% RSLogix 500 project I2P HANDS-ON 3 - LEO.RSS, saved by version 10.00.00.00 %
PROJECT "ML04B"    % processor: Bul.1763 MicroLogix 1100 Series B %

PROGRAM FILES
  LAD 2   10 rungs

DATA FILES
  O0 OUTPUT  4 elements
  I1 INPUT  6 elements
  S2 STATUS  66 elements
  B3 BINARY  1 elements
  T4 TIMER  1 elements
  C5 COUNTER  1 elements
  R6 CONTROL  1 elements
  N7 INTEGER  1 elements
  F8 FLOAT  1 elements

LADDER 2
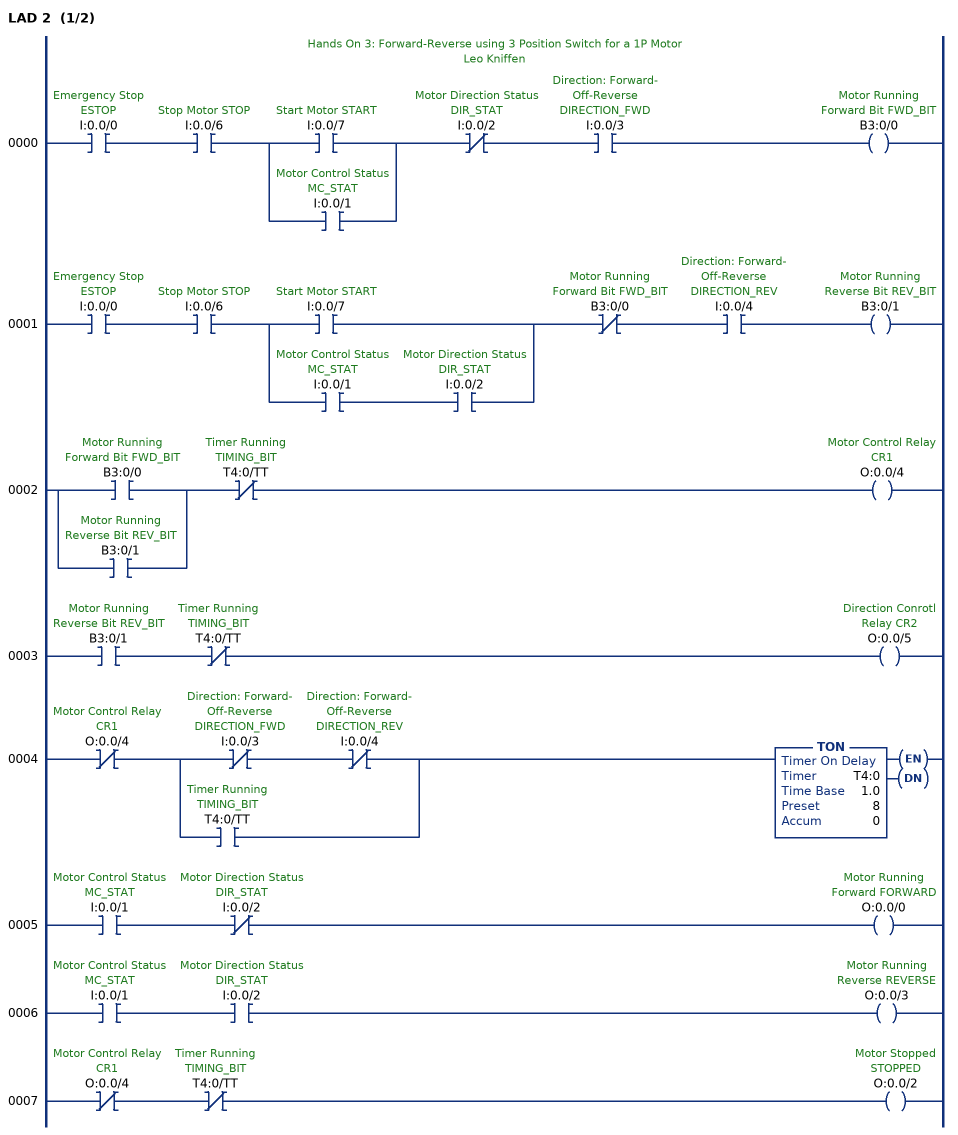
% Rung: 0 %
% Hands On 3: Forward-Reverse using 3 Position Switch for a 1P Motor
% Leo Kniffen %
SOR XIC I:0.0/0 XIC I:0.0/6 BST XIC I:0.0/7 NXB XIC I:0.0/1 BND XIO I:0.0/2 XIC I:0.0/3 OTE B3:0/0 EOR
%   I:0.0/0  ESTOP  "Emergency Stop" %
%   I:0.0/6  STOP  "Stop Motor" %
%   I:0.0/7  START  "Start Motor" %
%   I:0.0/1  MC_STAT  "Motor Control Status" %
%   I:0.0/2  DIR_STAT  "Motor Direction Status" %
%   I:0.0/3  DIRECTION_FWD  "Direction: Forward- Off-Reverse" %
%   B3:0/0  FWD_BIT  "Motor Running Forward Bit" %
% Rung: 1 %
SOR XIC I:0.0/0 XIC I:0.0/6 BST XIC I:0.0/7 NXB XIC I:0.0/1 XIC I:0.0/2 BND XIO B3:0/0 XIC I:0.0/4 OTE B3:0/1 EOR
%   I:0.0/0  ESTOP  "Emergency Stop" %
%   I:0.0/6  STOP  "Stop Motor" %
%   I:0.0/7  START  "Start Motor" %
%   I:0.0/1  MC_STAT  "Motor Control Status" %
%   I:0.0/2  DIR_STAT  "Motor Direction Status" %
%   B3:0/0  FWD_BIT  "Motor Running Forward Bit" %
%   I:0.0/4  DIRECTION_REV  "Direction: Forward- Off-Reverse" %
%   B3:0/1  REV_BIT  "Motor Running Reverse Bit" %
% Rung: 2 %
SOR BST XIC B3:0/0 NXB XIC B3:0/1 BND XIO T4:0/TT OTE O:0.0/4 EOR
%   B3:0/0  FWD_BIT  "Motor Running Forward Bit" %
%   B3:0/1  REV_BIT  "Motor Running Reverse Bit" %
%   T4:0/TT  TIMING_BIT  "Timer Running" %
%   O:0.0/4  CR1  "Motor Control Relay" %
% Rung: 3 %
SOR XIC B3:0/1 XIO T4:0/TT OTE O:0.0/5 EOR
%   B3:0/1  REV_BIT  "Motor Running Reverse Bit" %
%   T4:0/TT  TIMING_BIT  "Timer Running" %
%   O:0.0/5  CR2  "Direction Conrotl Relay" %
% Rung: 4 %
SOR XIO O:0.0/4 BST XIO I:0.0/3 XIO I:0.0/4 NXB XIC T4:0/TT BND TON T4:0 1.0 8 0 EOR
%   O:0.0/4  CR1  "Motor Control Relay" %
%   I:0.0/3  DIRECTION_FWD  "Direction: Forward- Off-Reverse" %
%   I:0.0/4  DIRECTION_REV  "Direction: Forward- Off-Reverse" %
%   T4:0/TT  TIMING_BIT  "Timer Running" %
% Rung: 5 %
SOR XIC I:0.0/1 XIO I:0.0/2 OTE O:0.0/0 EOR
%   I:0.0/1  MC_STAT  "Motor Control Status" %
%   I:0.0/2  DIR_STAT  "Motor Direction Status" %
%   O:0.0/0  FORWARD  "Motor Running Forward" %
% Rung: 6 %
SOR XIC I:0.0/1 XIC I:0.0/2 OTE O:0.0/3 EOR
%   I:0.0/1  MC_STAT  "Motor Control Status" %
%   I:0.0/2  DIR_STAT  "Motor Direction Status" %
%   O:0.0/3  REVERSE  "Motor Running Reverse" %
% Rung: 7 %
SOR XIO O:0.0/4 XIO T4:0/TT OTE O:0.0/2 EOR
%   O:0.0/4  CR1  "Motor Control Relay" %
%   T4:0/TT  TIMING_BIT  "Timer Running" %
%   O:0.0/2  STOPPED  "Motor Stopped" %

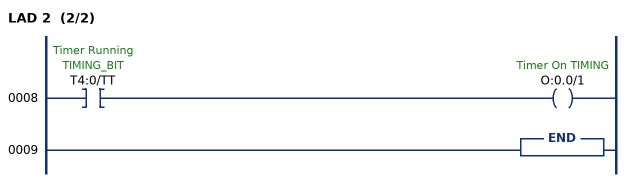
% Rung: 8 %
SOR XIC T4:0/TT OTE O:0.0/1 EOR
%   T4:0/TT  TIMING_BIT  "Timer Running" %
%   O:0.0/1  TIMING  "Timer On" %
% Rung: 9 %
SOR END EOR

DATA TABLE (non-zero values as saved)
DATA T4
% .PRE .ACC %
% T4:0 % 8 0
